// TIA Portal V19 export
FUNCTION_BLOCK "TYPIC_C501_IF_KLG"   // FB64, FBD
TITLE = TYPIC_C501_IF_KLG: Motorgestuurde klep
{ S7_Optimized_Access := 'TRUE' }
AUTHOR : OCOTECH
FAMILY : Typical
NAME : C501.703
// Logisch Object Besturing: C501.703
// 
// De interne functie motorgestuurde klep verzorgt de interne besturing, bewaking en fysieke aansturing van een motorgestuurde klep behorend tot de brandblusinstallatie.
// stored: MemoryReserve 10, SetENOAutomatically false
   VAR_INPUT
      EXT_HW { ExternalAccessible := 'False'; ExternalVisible := 'False'; ExternalWritable := 'False'} : Bool;   // Sturings hardware (PLC) bewaking (1 = OK)
      IN_OPEN { ExternalAccessible := 'False'; ExternalVisible := 'False'; ExternalWritable := 'False'} : Bool;   // Klep is open
      IN_TOE { ExternalAccessible := 'False'; ExternalVisible := 'False'; ExternalWritable := 'False'} : Bool;   // Klep is toe
      IN_AUT_C501 { ExternalAccessible := 'False'; ExternalVisible := 'False'; ExternalWritable := 'False'} : Bool;   // Beveiligingen: serie geschakelde terugmelding (1= OK)
      CFG_TYD_FB { ExternalAccessible := 'False'; ExternalVisible := 'False'; ExternalWritable := 'False'} : Time;   // Vertragingstijd storing foute terugmelding
   END_VAR
   VAR_OUTPUT
      VAR_IF_KLG { ExternalAccessible := 'False'; ExternalVisible := 'False'; ExternalWritable := 'False'} : "C501_VAR_IF_KLG_TYPIC";   // Struct met alle variabelen naar bovenliggende functies
      OUT_OPEN { ExternalAccessible := 'False'; ExternalVisible := 'False'; ExternalWritable := 'False'} : Bool;   // Klep openen
      OUT_TOE { ExternalAccessible := 'False'; ExternalVisible := 'False'; ExternalWritable := 'False'} : Bool;   // Klep sluiten
   END_VAR
   VAR_IN_OUT
      STU_IF_KLG : "C501_STU_IF_KLG_TYPIC";   // Struct met alle sturingen van de subfunctie (SF) motorgestuurde klep van 3B
   END_VAR
   VAR
      BED : Struct   // Bedieningen
         REM : Bool;   // Bediening om klep in Remote te schakelen (indien IN_HND = 0)
         OPEN : Bool;   // Bediening om klep in hand te schakelen en te openen
         TOE : Bool;   // Bediening om klep in hand te schakelen en te sluiten
         RES : Bool;   // Reset storingen
      END_STRUCT;
      STO { ExternalWritable := 'False'} : Struct   // Storingen
         A001 : Bool;   // Beveiliging aangesproken
         AT01 : Bool;   // Terugmelding Open niet ontvangen
         AT02 : Bool;   // Terugmelding Dicht niet ontvangen
         AT03 : Bool;   // Terugmeldingen Open en Dicht tegelijkertijd
      END_STRUCT;
      VAR { ExternalWritable := 'False'} : Struct   // Variabelen
         HAND_OPEN { ExternalAccessible := 'False'; ExternalVisible := 'False'} : Bool;   // TRUE = Gewenste stand in hand is Open FALSE = Gewenste stand in hand is Toe
         CMD_OPEN { ExternalAccessible := 'False'; ExternalVisible := 'False'} : Bool;   // TRUE = Gewenste stand is Open FALSE = Gewenste stand is Toe
         STS_OPEN : Bool;   // Motorgestuurde klep is open
         STS_TOE : Bool;   // Motorgestuurde klep is toe
         STS_BEZ_OPEN : Bool;   // Motorgestuurde klep is aan het openen (1 = Open)
         STS_BEZ_TOE : Bool;   // Motorgestuurde klep is aan het sluiten (1 = Toe)
         BMO_HAND : Bool;   // TRUE = in hand geschakeld FALSE = niet in hand
         EXT_HW { ExternalAccessible := 'False'; ExternalVisible := 'False'} : Bool;   // Sturings hardware (PLC) in storing
      END_STRUCT;
   END_VAR
BEGIN

REGION Network 1: START
END_REGION

REGION Network 2: +++ Werkingsmode Hand +++
   // Verwerking van de bedieningen van het aanraakscherm, en bepalen van de bedieningsmode Hand.
END_REGION

REGION Network 3: +++ Gewenste stand +++
   // Bepalen aan de hand van de actuele bediening of ontvangen sturing, wat de gewenste stand van de klep is.
END_REGION

REGION Network 4: +++ Klepsturing +++
   // Aansturen van de klep en terugmeldingsbewaking.
END_REGION

REGION Network 5: +++ Storingen +++
   // Verwerken van de storingsmeldingen.
END_REGION

REGION Network 6: Storing A001: Beveiliging aangesproken
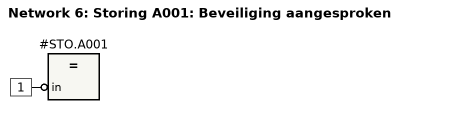
   #STO.A001 := NOT 1;
END_REGION

REGION Network 7 (SCL): EINDE
   // Variabelen van intern scada rakvlak naar outputs copieren
   #VAR_IF_KLG.STS_OPEN := #VAR.STS_OPEN;
   #VAR_IF_KLG.STS_TOE := #VAR.STS_TOE;
   #VAR_IF_KLG.STS_BEZ_OPEN := #VAR.STS_BEZ_OPEN;
   #VAR_IF_KLG.STS_BEZ_TOE := #VAR.STS_BEZ_TOE;
   #VAR_IF_KLG.BMO_HAND := #VAR.BMO_HAND;
   #VAR_IF_KLG.EXT_HW := #VAR.EXT_HW;
   #VAR_IF_KLG.STO := #STO;
END_REGION
END_FUNCTION_BLOCK
